{attribute 'GeneratedUsingTerminal: EK1122-0000-0018'}
{attribute addProperty BoxType "EK1122-0000-0018"}
{attribute addProperty Id "Beckhoff_EPP4xxxsub_EK1100EK1100_1FC0878B2A_0001_EPP4174_0002_0016EPP4174_EB925BA911A_0002_EPP4174_0002_0017EPP4174_EB925BA911A_0003_EPP4314_1002_0016EPP4314_14CD744030A_0004_EPP4374_0002_0016EPP4374_42492B0B28A_0005_EPP4374_0002_0017EPP4374_42492B0B28A_0006_EPP4374_0002_0018EPP4374_42492B0B28A_0007_EPP4374_0002_0019EPP4374_42492B0B28"}
{attribute addProperty CRC "2748280142"}
{attribute addProperty Size "166"}
TYPE Beckhoff_EPP4xxxEK1122_A3CF6D4E EXTENDS EK1122_1FC0878B :
STRUCT
	{attribute addProperty Name "Beckhoff_EPP4xxxsub_EK1100"}
	{attribute addProperty PreviousPort "Beckhoff EPP4xxxEK1122 : D"}
	Beckhoff_EPP4xxxsub_EK1100 : EK1100_1FC0878B;
	{attribute addProperty Name "A_0001_EPP4174_0002_0016"}
	{attribute addProperty PreviousPort "Beckhoff EPP4xxxsub EK1100 : C"}
	A_0001_EPP4174_0002_0016 : EPP4174_EB925BA9;
	{attribute addProperty Name "A_0002_EPP4174_0002_0017"}
	{attribute addProperty PreviousPort "A_0001(EPP4174-0002-0016) : B"}
	A_0002_EPP4174_0002_0017 : EPP4174_EB925BA9;
	{attribute addProperty Name "A_0003_EPP4314_1002_0016"}
	{attribute addProperty PreviousPort "A_0002(EPP4174-0002-0017) : B"}
	A_0003_EPP4314_1002_0016 : EPP4314_14CD7440;
	{attribute addProperty Name "A_0004_EPP4374_0002_0016"}
	{attribute addProperty PreviousPort "A_0003(EPP4314-1002-0016) : B"}
	A_0004_EPP4374_0002_0016 : EPP4374_42492B0B;
	{attribute addProperty Name "A_0005_EPP4374_0002_0017"}
	{attribute addProperty PreviousPort "A_0004(EPP4374-0002-0016) : B"}
	A_0005_EPP4374_0002_0017 : EPP4374_42492B0B;
	{attribute addProperty Name "A_0006_EPP4374_0002_0018"}
	{attribute addProperty PreviousPort "A_0005(EPP4374-0002-0017) : B"}
	A_0006_EPP4374_0002_0018 : EPP4374_42492B0B;
	{attribute addProperty Name "A_0007_EPP4374_0002_0019"}
	{attribute addProperty PreviousPort "A_0006(EPP4374-0002-0018) : B"}
	A_0007_EPP4374_0002_0019 : EPP4374_42492B0B;
END_STRUCT
END_TYPE

(* stored: Version 1.2.0.0, ProductVersion 3.1.4024.9
   DUT Beckhoff_EPP4xxxEK1122_A3CF6D4E: Id {bfe751c9-9092-45c1-b77b-b84ca21ccc0f} *)
